FUNCTION_BLOCK E_TOF (* standard timer function block (off-delay timing) *)
  (* Standard: 61499-2; Classification: standard timer function block; Description: Copyright (c) 2024 HR Agrartechnik GmbH This program and the accompanying materials are made available under the terms of the Eclipse Public License 2.0 which is available at https://www.eclipse.org/legal/epl-2.0/ SPDX-License-Identifier: EPL-2.0 *)
  (* Version 1.0, 2024-03-04, Franz Hoepfinger, HR Agrartechnik GmbH *)
  (* Version 1.1, 2024-04-23, Franz Hoepfinger, HR Agrartechnik GmbH, Add a Reset to Timer FBs *)
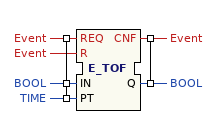
  EVENT_INPUT
    REQ WITH IN, PT; (* Normal Execution Request *)
    R; (* Reset *)
  END_EVENT
  EVENT_OUTPUT
    CNF WITH Q; (* Execution Confirmation *)
  END_EVENT
  VAR_INPUT
    IN : BOOL; (* Input *)
    PT : TIME; (* Process time *)
  END_VAR
  VAR_OUTPUT
    Q : BOOL; (* Output *)
  END_VAR
  FBS
    E_SWITCH : E_SWITCH;
    E_DELAY : E_DELAY;
    E_RS : E_RS;
  END_FBS
  EVENT_CONNECTIONS
    REQ TO E_SWITCH.EI;
    E_RS.EO TO CNF;
    E_DELAY.EO TO E_RS.R;
    E_SWITCH.EO1 TO E_RS.S;
    E_SWITCH.EO0 TO E_DELAY.START;
    E_SWITCH.EO1 TO E_DELAY.STOP;
    R TO E_RS.R;
    R TO E_DELAY.STOP;
  END_CONNECTIONS
  DATA_CONNECTIONS
    IN TO E_SWITCH.G;
    PT TO E_DELAY.DT;
    E_RS.Q TO Q;
  END_CONNECTIONS
END_FUNCTION_BLOCK
